// TwinCAT 3 PLC project core
// Title: Nepionic Core
// Company: Nepionic
// Author: Nepionic
// ProjectVersion: 0.1.0
// ProgramVersion: 3.1.4026.16
// project tree:
//   commands/AsyncCommand/ NoopAsyncCommand.TcPOU, AsyncCommand.TcIO
//   commands/AsyncCommand/Runners/ SingleAsyncCommandRunner.TcPOU
//   commands/Command/ I_Command.TcIO
//   commands/Internal/AsyncCommandStateMachine/ AsyncCommandStateMachine.TcPOU, AsyncCommandStateControl.TcIO
//   disposable/ DefaultDisposable.TcPOU, Disposable.TcIO

// ---- commands/AsyncCommand/AsyncCommand.TcIO
INTERFACE PUBLIC AsyncCommand EXTENDS I_Command

METHOD PUBLIC Abort
END_METHOD

PROPERTY PUBLIC Busy : BOOL
GET
END_GET
END_PROPERTY

METHOD PUBLIC CyclicCall
END_METHOD

PROPERTY PUBLIC Done : BOOL
GET
END_GET
END_PROPERTY

PROPERTY PUBLIC Error : BOOL
GET
END_GET
END_PROPERTY

PROPERTY PUBLIC ErrorId : UDINT
GET
END_GET
END_PROPERTY

END_INTERFACE

// ---- commands/Command/I_Command.TcIO
INTERFACE PUBLIC I_Command EXTENDS Disposable

METHOD PUBLIC Execute
END_METHOD

END_INTERFACE

// ---- commands/Internal/AsyncCommandStateMachine/AsyncCommandStateControl.TcIO
INTERFACE AsyncCommandStateControl

METHOD PUBLIC Error
VAR_INPUT
	ErrorId : UDINT;
END_VAR
END_METHOD

METHOD PUBLIC Next
VAR_INPUT
END_VAR
END_METHOD

END_INTERFACE

// ---- disposable/Disposable.TcIO
INTERFACE Disposable EXTENDS __System.IQueryInterface

METHOD PUBLIC Dispose
END_METHOD

END_INTERFACE

// ---- commands/AsyncCommand/NoopAsyncCommand.TcPOU
{attribute 'linkalways'} 
{attribute 'no_explicit_call' := 'This FB is a CLASS and must be accessed using methods or properties'}
{attribute 'enable_dynamic_creation'}
FUNCTION_BLOCK PUBLIC NoopAsyncCommand EXTENDS DefaultDisposable IMPLEMENTS AsyncCommand
VAR
	state_machine : AsyncCommandStateMachine;
END_VAR

METHOD PUBLIC Abort
state_machine.Abort();
END_METHOD

PROPERTY PUBLIC Busy : BOOL
GET // PUBLIC
IF state_machine.IsAborted THEN
	RETURN;
END_IF

IF state_machine.IsCompleted THEN
	RETURN;
END_IF

IF state_machine.IsErrored THEN
	RETURN;
END_IF

IF state_machine.IsIdle THEN
	RETURN;
END_IF

Busy := TRUE;
END_GET
END_PROPERTY

METHOD PUBLIC CyclicCall
IF state_machine.IsIdle THEN
	OnIdle();
END_IF

IF state_machine.IsInitializing THEN
	OnInitializing(state_machine);
END_IF

IF state_machine.IsExecuting THEN
	OnExecuting(state_machine);
END_IF

IF state_machine.IsCompleting THEN
	OnCompleting(state_machine);
END_IF

IF state_machine.IsCompleted THEN
	OnCompleted();
END_IF

IF state_machine.IsAborting THEN
	OnAborting(state_machine);
END_IF

IF state_machine.IsAborted THEN
	OnAborted();
END_IF

IF state_machine.IsErrored THEN
	OnErrored();
END_IF
END_METHOD

PROPERTY PUBLIC Done : BOOL
GET // PUBLIC
Done := state_machine.IsCompleted;
END_GET
END_PROPERTY

PROPERTY PUBLIC Error : BOOL
GET // PUBLIC
Error := state_machine.IsErrored;
END_GET
END_PROPERTY

PROPERTY PUBLIC ErrorId : UDINT
GET // PUBLIC
ErrorId := state_machine.ErrorId;
END_GET
END_PROPERTY

METHOD PUBLIC Execute
state_machine.Execute();
END_METHOD

METHOD PROTECTED OnAborted
END_METHOD

METHOD PROTECTED OnAborting
VAR_INPUT
	state_control : AsyncCommandStateControl;
END_VAR
// default behaviour is to go to next state
// you can override this method to implement your own completing control code.
// just call StateControl.Next() when your code is completed.  

state_control.Next();
END_METHOD

METHOD PROTECTED OnCompleted : BOOL
END_METHOD

METHOD PROTECTED OnCompleting
VAR_INPUT
	state_control : AsyncCommandStateControl;
END_VAR
// default behaviour is to go to next state
// you can override this method to implement your own completing control code.
// just call StateControl.Next() when your code is completed.  

state_control.Next();
END_METHOD

METHOD PROTECTED OnErrored
END_METHOD

METHOD PROTECTED OnExecuting
VAR_INPUT
	state_control : AsyncCommandStateControl;
END_VAR
// default behaviour is to go to next state
// you can override this method to implement your own executing control code.
// just call StateControl.Next() when your code is completed.  

state_control.Next();
END_METHOD

METHOD PROTECTED OnIdle
END_METHOD

METHOD PROTECTED OnInitializing
VAR_INPUT
	state_control : AsyncCommandStateControl;
END_VAR
// default behaviour is to go to next state
// you can override this method to implement your own initializing control code.
// just call StateControl.Next() when your code is completed.  

state_control.Next();
END_METHOD

END_FUNCTION_BLOCK

// ---- disposable/DefaultDisposable.TcPOU
{attribute 'linkalways'} 
{attribute 'no_explicit_call' := 'This FB is a CLASS and must be accessed using methods or properties'}
{attribute 'enable_dynamic_creation'}
FUNCTION_BLOCK ABSTRACT DefaultDisposable IMPLEMENTS Disposable

METHOD PUBLIC Dispose
VAR
	pDisposable : POINTER TO DefaultDisposable;
END_VAR
pDisposable := THIS;
__DELETE(pDisposable);
END_METHOD

METHOD FB_exit : BOOL
VAR_INPUT
	bInCopyCode : BOOL; // if TRUE, the exit method is called for exiting an instance that is copied afterwards (online change).
END_VAR
// by default you would return if this is an in copy code, i.e. online change to this class
IF bInCopyCode THEN
	RETURN;
END_IF

// A word of warning. FB_exit does not NOT operate in the same way as a typical inherited method. If a child class does not implement FB_exit then it does not
// gain this one for itself. 
// The system will automatically call each FB_exit on each layer of inheritance one by one, starting with the child class and making it's way to the parent.
// Therefore code in here will only be triggered once the system reaches this layer of the object's deletion. The child class and all of it's variables
// will already have had FB_exit called by the time we reach this point!
END_METHOD

END_FUNCTION_BLOCK

// ---- commands/Internal/AsyncCommandStateMachine/AsyncCommandStateMachine.TcPOU
{attribute 'linkalways'} 
{attribute 'no_explicit_call' := 'This FB is a CLASS and must be accessed using methods or properties'}
{attribute 'enable_dynamic_creation'}
FUNCTION_BLOCK INTERNAL AsyncCommandStateMachine IMPLEMENTS AsyncCommandStateControl
VAR
	state : (IDLE, INITIALIZING, EXECUTING, COMPLETING, COMPLETED, ABORTING, ABORTED, ERRORED);
	_errorId : UDINT;
END_VAR

METHOD PUBLIC Abort
VAR_INPUT
END_VAR
CASE state OF
	IDLE : RETURN;
	ABORTING : RETURN;
	COMPLETED : RETURN;
	ABORTED : RETURN;
	ERRORED : RETURN;
END_CASE

state := ABORTING;
END_METHOD

METHOD PUBLIC Error
VAR_INPUT
	ErrorId : UDINT;
END_VAR
CASE state OF
	IDLE : RETURN;
	COMPLETED : RETURN;
	ABORTED : RETURN;
	ERRORED : RETURN;
END_CASE

_errorId := ErrorId;
state := ERRORED;
END_METHOD

{attribute 'monitoring' := 'call'}
PROPERTY PUBLIC ErrorId : UDINT
GET
ErrorID := _errorId;
END_GET
END_PROPERTY

METHOD PUBLIC Execute
VAR_INPUT
END_VAR
CASE state OF
	INITIALIZING : RETURN;
	EXECUTING : RETURN;
	COMPLETING : RETURN;
	ABORTING : RETURN;
END_CASE

_errorId := 0;
state := INITIALIZING;
END_METHOD

{attribute 'monitoring' := 'call'}
PROPERTY PUBLIC IsAborted : BOOL
GET
IsAborted := state = ABORTED;
END_GET
END_PROPERTY

{attribute 'monitoring' := 'call'}
PROPERTY PUBLIC IsAborting : BOOL
GET
IsAborting := state = ABORTING;
END_GET
END_PROPERTY

{attribute 'monitoring' := 'call'}
PROPERTY PUBLIC IsCompleted : BOOL
GET
IsCompleted := state = COMPLETED;
END_GET
END_PROPERTY

{attribute 'monitoring' := 'call'}
PROPERTY PUBLIC IsCompleting : BOOL
GET
IsCompleting := state = COMPLETING;
END_GET
END_PROPERTY

{attribute 'monitoring' := 'call'}
PROPERTY PUBLIC IsErrored : BOOL
GET
IsErrored := state = ERRORED;
END_GET
END_PROPERTY

{attribute 'monitoring' := 'call'}
PROPERTY PUBLIC IsExecuting : BOOL
GET
IsExecuting := state = EXECUTING;
END_GET
END_PROPERTY

{attribute 'monitoring' := 'call'}
PROPERTY PUBLIC IsIdle : BOOL
GET
IsIdle:= state = IDLE;
END_GET
END_PROPERTY

{attribute 'monitoring' := 'call'}
PROPERTY PUBLIC IsInitializing : BOOL
GET
IsInitializing := state = INITIALIZING;
END_GET
END_PROPERTY

METHOD PUBLIC Next
VAR_INPUT
END_VAR
CASE state OF
	IDLE : RETURN;
	INITIALIZING : StateComplete_Initializing();
	EXECUTING : StateComplete_Executing();
	COMPLETING : StateComplete_Completing();
	COMPLETED : RETURN;
	ABORTING : StateComplete_Aborting();
	ABORTED : RETURN;
	ERRORED : RETURN;
END_CASE
END_METHOD

METHOD PRIVATE StateComplete_Aborting
VAR_INPUT
END_VAR
state := ABORTED;
END_METHOD

METHOD PRIVATE StateComplete_Completing
VAR_INPUT
END_VAR
state := COMPLETED;
END_METHOD

METHOD PRIVATE StateComplete_Executing
VAR_INPUT
END_VAR
state := COMPLETING;
END_METHOD

METHOD PRIVATE StateComplete_Initializing
VAR_INPUT
END_VAR
state := EXECUTING;
END_METHOD

END_FUNCTION_BLOCK

// ---- commands/AsyncCommand/Runners/SingleAsyncCommandRunner.TcPOU
{attribute 'linkalways'} 
{attribute 'no_explicit_call' := 'This FB is a CLASS and must be accessed using methods or properties'}
{attribute 'enable_dynamic_creation'}
FUNCTION_BLOCK PUBLIC SingleAsyncCommandRunner
VAR
	current_command : AsyncCommand;
	replacement_command : AsyncCommand;
END_VAR

PROPERTY PUBLIC Busy : BOOL
GET // PUBLIC
IF current_command = 0 THEN
	RETURN;
END_IF

Busy := current_command.Busy;
END_GET
END_PROPERTY

METHOD PUBLIC CyclicCall
IF current_command <> 0 AND_THEN current_command.Busy THEN
	current_command.CyclicCall();
	RETURN;
END_IF

IF replacement_command <> 0 THEN
	current_command := replacement_command;
	replacement_command := 0;
	current_command.Execute();
END_IF
END_METHOD

PROPERTY Done : BOOL
GET // PUBLIC
IF current_command = 0 THEN
	RETURN;
END_IF

Done := current_command.Done;
END_GET
END_PROPERTY

PROPERTY Error : BOOL
GET // PUBLIC
IF current_command = 0 THEN
	RETURN;
END_IF

Error := current_command.Error;
END_GET
END_PROPERTY

PROPERTY PUBLIC ErrorId : UDINT
GET // PUBLIC
IF current_command = 0 THEN
	RETURN;
END_IF

ErrorId := current_command.ErrorId;
END_GET
END_PROPERTY

METHOD ExecuteCommand
VAR_INPUT
	command : AsyncCommand;
END_VAR
IF current_command = 0 THEN
	current_command := command;
	current_command.Execute();
	RETURN;
END_IF

current_command.Abort();
replacement_command := command;
END_METHOD

END_FUNCTION_BLOCK
